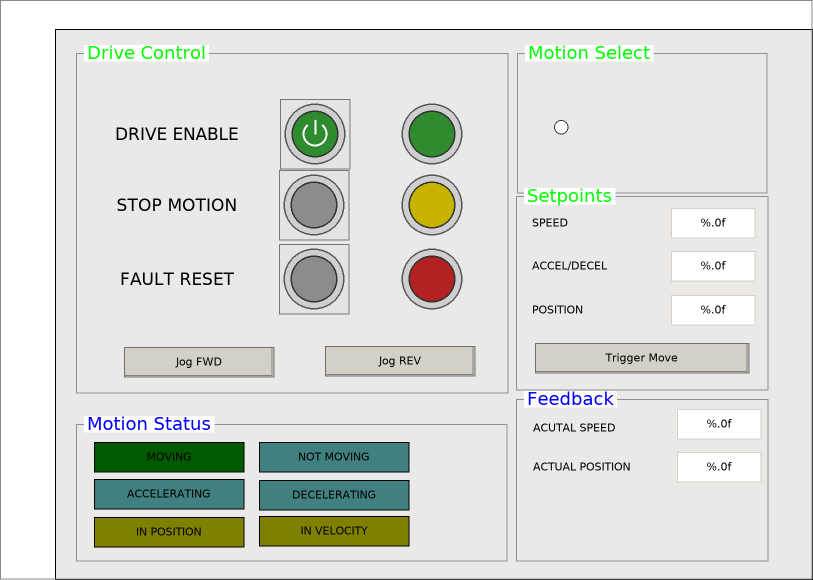
VISUALIZATION MotorFaceplate2  // 813x580
    Rectangle (55,29 758x551)
    GroupBox (76,45 432x348), "Drive Control"
        PowerSwitch (204,54 70x70), behaviour: TOGGLE, style: Switch-PowerSwitch-Green
        PushSwitch (203,125 70x70), behaviour: TOGGLE, style: Switch-PushSwitch-Gray
        PushSwitch (203,199 70x70), behaviour: TOGGLE, style: Switch-PushSwitch-Gray
        Lamp1 (321,54 70x70), style: Lamp-Lamp1-Green
        Lamp1 (321,125 70x70), style: Lamp-Lamp1-Yellow
        Lamp1 (321,199 70x70), style: Lamp-Lamp1-Red
        Label (26,74 150x30), "DRIVE ENABLE"
        Label (26,145 150x30), "STOP MOTION"
        Label (26,219 150x30), "FAULT RESET"
        Button (249,301 150x30), "Jog REV"
    GroupBox (517,45 250x148), "Motion Select"
        RadioButton (35,21 173x122), variable: ServoGVLs.servo1Interface.iMotionSelect
    GroupBox (516,188 252x202), "Setpoints"
        Label (13,20 76x30), "SPEED"
        Textfield (155,20 84x30), "%.0f"
        Label (13,63 99x30), "ACCEL/DECEL"
        Textfield (155,63 84x30), "%.0f"
        Label (13,107 76x30), "POSITION"
        Textfield (155,107 84x30), "%.0f"
        Button (19,155 214x30), "Trigger Move"
    GroupBox (76,416 431x145), "Motion Status"
        RoundedRectangle (18,26 150x30), "MOVING"
        RoundedRectangle (183,26 150x30), "NOT MOVING"
        RoundedRectangle (18,63 150x30), "ACCELERATING"
        RoundedRectangle (183,64 150x30), "DECELERATING"
        RoundedRectangle (18,101 150x30), "IN POSITION"
        RoundedRectangle (183,100 150x30), "IN VELOCITY"
    GroupBox (516,391 252x170), "Feedback"
        Textfield (161,18 84x30), "%.0f"
        Label (14,61 120x30), "ACTUAL POSITION"
        Textfield (161,61 84x30), "%.0f"
        Label (14,22 108x30), "ACUTAL SPEED"
    Button (124,347 150x30), "Jog FWD"
END_VISUALIZATION

(* stored: Version 1.1.0.1, ProductVersion 3.1.4024.12
   Visu MotorFaceplate2: Id {e0f65b2a-af48-4dbc-a903-34ea7d1fbc3e} *)
